{attribute 'GeneratedUsingTerminal: EL5151-0000-0016'}
{attribute addProperty BoxType "EL5151-0000-0016"}
{attribute addProperty Id "StatusAT %I*Status_396FCBA08Counter_valueAT %I*UDINT4Latch_valueAT %I*UDINT4"}
{attribute addProperty CRC "865715626"}
{attribute addProperty Size "16"}
TYPE ENC_Inputs_3399C5AA :
STRUCT
	{attribute addProperty Name "Status"}
	Status AT %I* : Status_396FCBA0;
	{attribute addProperty Name "Counter_value"}
	Counter_value AT %I* : UDINT;
	{attribute addProperty Name "Latch_value"}
	Latch_value AT %I* : UDINT;
END_STRUCT
END_TYPE

(* stored: Version 1.2.0.0, ProductVersion 3.1.4024.9
   DUT ENC_Inputs_3399C5AA: Id {a18cffbf-8f71-4aca-822a-746aa1997ac5} *)
